	FUNCTION_BLOCK FB 303
	TITLE =G203M COUPLING DEVICE TURNER GERM 6
	//COPYRIGHT:    (C) 2009  BUHLER AG, CH-9240 UZWIL, SWITZERLAND
	//
	//PRODUCT:      WinCoS_BIW01_09
	//
	//TITLE:        COUPLING DEVICE TURNER GERM 6
	//                Machine group control
	//                Maschinengruppensteuerung
	//
	//--------------------------------------------------------------------------------
	//
	//IDENT:        AUTHOR:             DEPT:                              DATE:
	//
	//P01_FB303.1.0 K.Renz              CSB41                              13.Jan.2010
	//             1st Release
	//
	//--------------------------------------------------------------------------------
	//
	//PURPOSE:
	//
	//MANUAL :
	//
	//RESTRICTIONS:
	//
	//--------------------------------------------------------------------------------
	AUTHOR  : KR
	FAMILY  : USW
	VERSION : 9.9


	VAR
	  Gr       : FB10;	//Standard interface to group
	  InOutValue1    : DINT; //Data for user
	  InOutValue2    : DINT; //Data for user
	  OutWayConflict : BOOL;	//Data for user
	  OutSelectionOk : BOOL;	//Data for user
	  CmdNewValue : BOOL;	//Data for user
	  CmdNewJob   : BOOL;	//Data for user
	  OutCodeOK   : BOOL;	//Data for user
	  InEndOfJob  : BOOL ;	//Data for user
	  staWayOk      : BOOL ;	//Data for user
	  EdgeStartRelease : BOOL ;	//Data for user
	  USW8  : BOOL;	//Data for user
	  USW9 : BOOL;	//Data for user
	  USW10: BOOL;	//Data for user
	  USW11: BOOL;	//Data for user
	  USW12: BOOL;	//Data for user
	  USW13: BOOL;	//Data for user
	  USW14: BOOL;	//Data for user
	  USW15: BOOL;	//Data for user
	     #A_2611_MXZ21 : FB12;   // Motor
	     #A_2611_BZS22 : FB14;   // DigInpCont
	     #A_2611_BZS23 : FB14;   // DigInpCont
	     #A_2611_MXZ25 : FB12;   // Motor
	     #A_2611_BZS26 : FB14;   // DigInpCont
	     #A_2611_BZS27 : FB14;   // DigInpCont
	     #A_2611_MXZ31 : FB12;   // Motor
	     #A_2611_BZS32 : FB14;   // DigInpCont
	     #A_2611_BZS33 : FB14;   // DigInpCont
	     #A_2611_MXZ35 : FB12;   // Motor
	     #A_2611_BZS36 : FB14;   // DigInpCont
	     #A_2611_BZS37 : FB14;   // DigInpCont
	END_VAR
	VAR_TEMP
	   tmpEnable		: BOOL;
	   tmpFlag  		: BOOL;
	   tmpCmdNext		: BOOL;
	   tmpLocal  		: BOOL;
	   tmpAspOk  		: BOOL;
	   tmpHWStop 		: BOOL;
	   tmpInstanzDBNo       : INT ;
	END_VAR
	BEGIN
	NETWORK
	TITLE =
	NETWORK
	TITLE =Read command from group control
	//Parameter
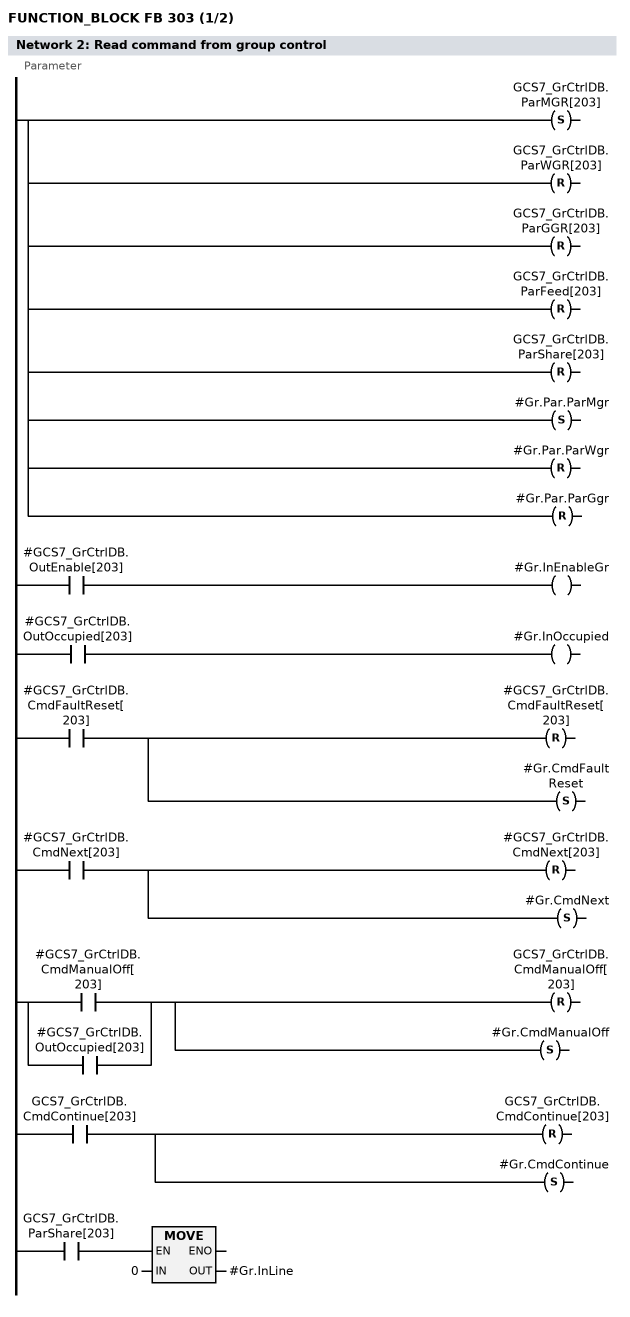
	      SET;
	      S   GCS7_GrCtrlDB.ParMGR[203];
	      R   GCS7_GrCtrlDB.ParWGR[203];
	      R   GCS7_GrCtrlDB.ParGGR[203];
	      R   GCS7_GrCtrlDB.ParFeed[203];
	      R   GCS7_GrCtrlDB.ParShare[203];
	      S   #Gr.Par.ParMgr;
	      R   #Gr.Par.ParWgr;
	      R   #Gr.Par.ParGgr;
	//Command
	      U   #GCS7_GrCtrlDB.OutEnable[203];
	      =   #Gr.InEnableGr;
	      U   #GCS7_GrCtrlDB.OutOccupied[203];
	      =   #Gr.InOccupied;
	      U   #GCS7_GrCtrlDB.CmdFaultReset[203];
	      R   #GCS7_GrCtrlDB.CmdFaultReset[203];
	      S   #Gr.CmdFaultReset;
	      U  #GCS7_GrCtrlDB.CmdNext[203];
	      R   #GCS7_GrCtrlDB.CmdNext[203];
	      S   #Gr.CmdNext;
	      U   #GCS7_GrCtrlDB.CmdManualOff[203];
	      O   #GCS7_GrCtrlDB.OutOccupied[203];
	      R   GCS7_GrCtrlDB.CmdManualOff[203];
	      S   #Gr.CmdManualOff;
	      U  GCS7_GrCtrlDB.CmdContinue[203];
	      R   GCS7_GrCtrlDB.CmdContinue[203];
	      S   #Gr.CmdContinue;
	//Init Line Number
	      U   GCS7_GrCtrlDB.ParShare[203];
	      SPBN WE00;
	      L     0;
	      T     #Gr.InLine;
	WE00: NOP   0;
	NETWORK
	TITLE =Call Methode Control
	// 1. Handle Interface PCControl
	// 2. Prepare mode --> ModePassive,ModeActive,ModeIdling
	// 3. Reset global flags of the group
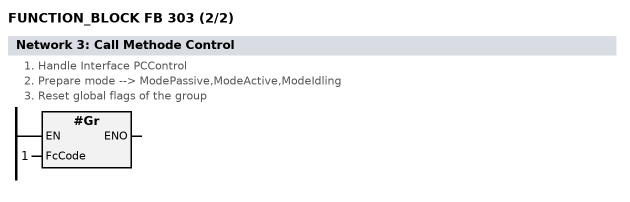
	      CALL #Gr (
	           FcCode                   := 1);
	NETWORK
	TITLE =Restart Idling Time
		L  #Gr.Par.ParIdling;
		L  2;
		>=I;
		SPB IdTm;
		T  #Gr.Par.ParIdling;
	IdTm:   NOP 0;
	      CLR;
	      S    #Gr.CmdRestartIdling;
	NETWORK
	TITLE =Prepare global flags
	NETWORK
	TITLE =Set Pattern (Target position)
	NETWORK
	TITLE =Interlocking WayOk
	//
	NETWORK
	TITLE =Interlocking Autostart
		CLR;
		R   #Gr.OutAutostart;
	NETWORK
	TITLE =Interlocking Enable
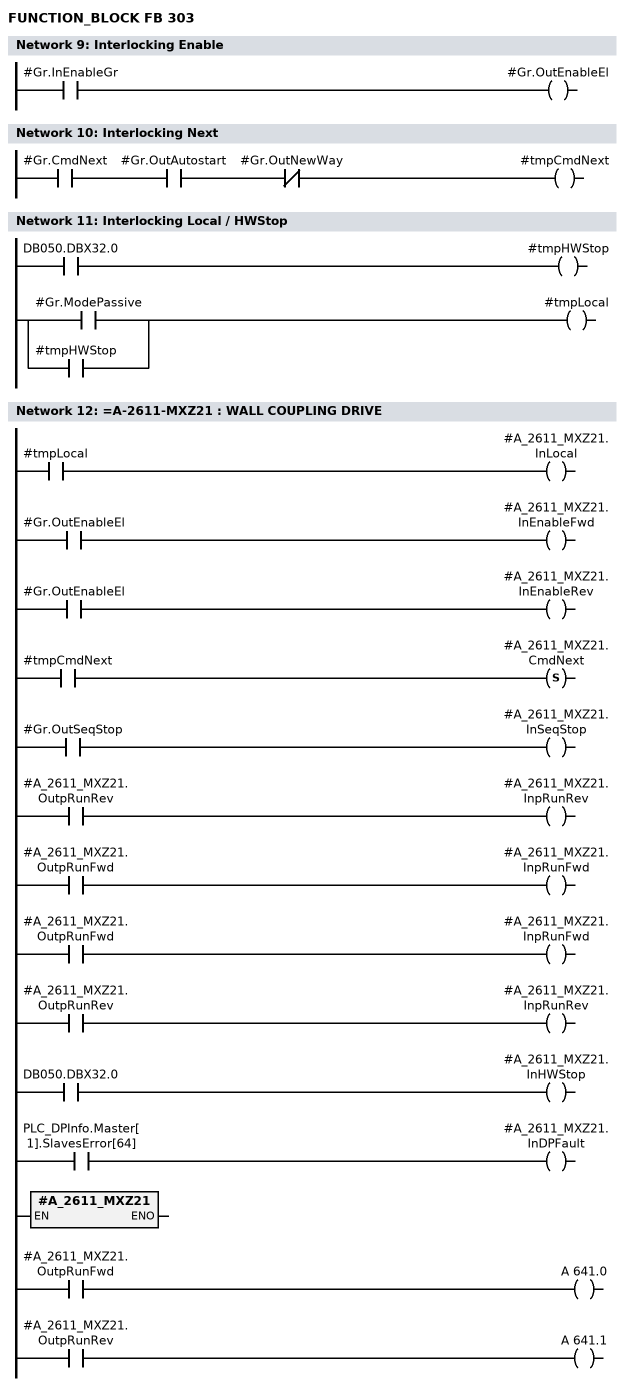
	      U     #Gr.InEnableGr;
	      =     #Gr.OutEnableEl;

	NETWORK
	TITLE =Interlocking Next
	      U     #Gr.CmdNext;
	      U     #Gr.OutAutostart;
	      UN    #Gr.OutNewWay;
	      =    #tmpCmdNext;

	NETWORK
	TITLE =Interlocking Local / HWStop
	      U    DB050.DBX32.0;
	      =    #tmpHWStop;

	      U    #Gr.ModePassive;
	      O    #tmpHWStop;
	      =    #tmpLocal;

	NETWORK
	TITLE ==A-2611-MXZ21 : WALL COUPLING DRIVE
	NOP 0;
	//-InLocal---
	      U     #tmpLocal;
	      =     #A_2611_MXZ21.InLocal;
	//
	//-Interlocking---
	      U     #Gr.OutEnableEl;
	      =     #A_2611_MXZ21.InEnableFwd;
	      U     #Gr.OutEnableEl;
	      =     #A_2611_MXZ21.InEnableRev;
	//
	      U    #tmpCmdNext;
	      S     #A_2611_MXZ21.CmdNext;
	//
	      U     #Gr.OutSeqStop;
	      =     #A_2611_MXZ21.InSeqStop;
	//
	//-Read inputs---
	      U     #A_2611_MXZ21.OutpRunRev;
	      =     #A_2611_MXZ21.InpRunRev;
	      U     #A_2611_MXZ21.OutpRunFwd;
	      =     #A_2611_MXZ21.InpRunFwd;
	      U     #A_2611_MXZ21.OutpRunFwd;
	      =     #A_2611_MXZ21.InpRunFwd;
	      U     #A_2611_MXZ21.OutpRunRev;
	      =     #A_2611_MXZ21.InpRunRev;
	      U   DB050.DBX32.0;
	      =     #A_2611_MXZ21.InHWStop;
	       U     PLC_DPInfo.Master[1].SlavesError[64];
	       =       #A_2611_MXZ21.InDPFault;
	//
	//-Set Parameters---
	//
	//-Call object control---
	      CALL  #A_2611_MXZ21;
	//
	//-Write outputs---
	      U     #A_2611_MXZ21.OutpRunFwd;
	      =     A 641.0;
	      U     #A_2611_MXZ21.OutpRunRev;
	      =     A 641.1;
	NETWORK
	TITLE ==A-2611-BZS22 : COUPLING DRIVE UNLOCKED
	NOP 0;
	//-InLocal---
	      U     #tmpLocal;
	      =     #A_2611_BZS22.InLocal;
	//
	//-Monitoring---
	      CLR;
	      =      #A_2611_BZS22.InMonTrue;
	      CLR;
	      =      #A_2611_BZS22.InMonFalse;
	//
	//-PreAlarm---
	      CLR;
	      =      #A_2611_BZS22.InPreAlarmTrue;
	      CLR;
	      =      #A_2611_BZS22.InPreAlarmFalse;
	//
	//-Additional commands---
	//      CLR
	//      S     #A_2611_BZS22.CmdRunTimeOutTime
	//
	//-Read inputs---
	      U     E 643.0;
	      =     #A_2611_BZS22.InpTrue;
	      U   DB050.DBX32.0;
	      =     #A_2611_BZS22.InHWStop;
	       U     PLC_DPInfo.Master[1].SlavesError[64];
	       =       #A_2611_BZS22.InDPFault;
	//
	//-Set Parameters---
	//
	//-Call object control---
	      CALL  #A_2611_BZS22;
	//
	//-Write outputs---
	NETWORK
	TITLE ==A-2611-BZS23 : COUPLING DRIVE LOCKED
	NOP 0;
	//-InLocal---
	      U     #tmpLocal;
	      =     #A_2611_BZS23.InLocal;
	//
	//-Monitoring---
	      CLR;
	      =      #A_2611_BZS23.InMonTrue;
	      CLR;
	      =      #A_2611_BZS23.InMonFalse;
	//
	//-PreAlarm---
	      CLR;
	      =      #A_2611_BZS23.InPreAlarmTrue;
	      CLR;
	      =      #A_2611_BZS23.InPreAlarmFalse;
	//
	//-Additional commands---
	//      CLR
	//      S     #A_2611_BZS23.CmdRunTimeOutTime
	//
	//-Read inputs---
	      U     E 643.1;
	      =     #A_2611_BZS23.InpTrue;
	      U   DB050.DBX32.0;
	      =     #A_2611_BZS23.InHWStop;
	       U     PLC_DPInfo.Master[1].SlavesError[64];
	       =       #A_2611_BZS23.InDPFault;
	//
	//-Set Parameters---
	//
	//-Call object control---
	      CALL  #A_2611_BZS23;
	//
	//-Write outputs---
	NETWORK
	TITLE ==A-2611-MXZ25 : WALL COUPLING DRIVE
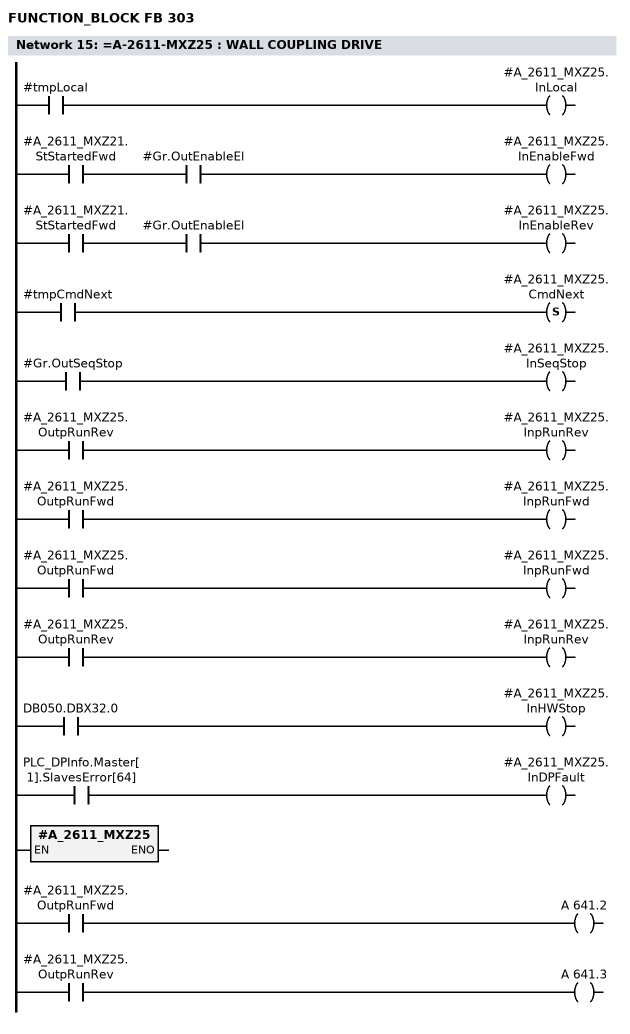
	NOP 0;
	//-InLocal---
	      U     #tmpLocal;
	      =     #A_2611_MXZ25.InLocal;
	//
	//-Interlocking---
	      U     #A_2611_MXZ21.StStartedFwd;
	      U     #Gr.OutEnableEl;
	      =     #A_2611_MXZ25.InEnableFwd;
	      U     #A_2611_MXZ21.StStartedFwd;
	      U     #Gr.OutEnableEl;
	      =     #A_2611_MXZ25.InEnableRev;
	//
	      U    #tmpCmdNext;
	      S     #A_2611_MXZ25.CmdNext;
	//
	      U     #Gr.OutSeqStop;
	      =     #A_2611_MXZ25.InSeqStop;
	//
	//-Read inputs---
	      U     #A_2611_MXZ25.OutpRunRev;
	      =     #A_2611_MXZ25.InpRunRev;
	      U     #A_2611_MXZ25.OutpRunFwd;
	      =     #A_2611_MXZ25.InpRunFwd;
	      U     #A_2611_MXZ25.OutpRunFwd;
	      =     #A_2611_MXZ25.InpRunFwd;
	      U     #A_2611_MXZ25.OutpRunRev;
	      =     #A_2611_MXZ25.InpRunRev;
	      U   DB050.DBX32.0;
	      =     #A_2611_MXZ25.InHWStop;
	       U     PLC_DPInfo.Master[1].SlavesError[64];
	       =       #A_2611_MXZ25.InDPFault;
	//
	//-Set Parameters---
	//
	//-Call object control---
	      CALL  #A_2611_MXZ25;
	//
	//-Write outputs---
	      U     #A_2611_MXZ25.OutpRunFwd;
	      =     A 641.2;
	      U     #A_2611_MXZ25.OutpRunRev;
	      =     A 641.3;
	NETWORK
	TITLE ==A-2611-BZS26 : COUPLING DRIVE UNLOCKED
	NOP 0;
	//-InLocal---
	      U     #tmpLocal;
	      =     #A_2611_BZS26.InLocal;
	//
	//-Monitoring---
	      CLR;
	      =      #A_2611_BZS26.InMonTrue;
	      CLR;
	      =      #A_2611_BZS26.InMonFalse;
	//
	//-PreAlarm---
	      CLR;
	      =      #A_2611_BZS26.InPreAlarmTrue;
	      CLR;
	      =      #A_2611_BZS26.InPreAlarmFalse;
	//
	//-Additional commands---
	//      CLR
	//      S     #A_2611_BZS26.CmdRunTimeOutTime
	//
	//-Read inputs---
	      U     E 643.2;
	      =     #A_2611_BZS26.InpTrue;
	      U   DB050.DBX32.0;
	      =     #A_2611_BZS26.InHWStop;
	       U     PLC_DPInfo.Master[1].SlavesError[64];
	       =       #A_2611_BZS26.InDPFault;
	//
	//-Set Parameters---
	//
	//-Call object control---
	      CALL  #A_2611_BZS26;
	//
	//-Write outputs---
	NETWORK
	TITLE ==A-2611-BZS27 : COUPLING DRIVE LOCKED
	NOP 0;
	//-InLocal---
	      U     #tmpLocal;
	      =     #A_2611_BZS27.InLocal;
	//
	//-Monitoring---
	      CLR;
	      =      #A_2611_BZS27.InMonTrue;
	      CLR;
	      =      #A_2611_BZS27.InMonFalse;
	//
	//-PreAlarm---
	      CLR;
	      =      #A_2611_BZS27.InPreAlarmTrue;
	      CLR;
	      =      #A_2611_BZS27.InPreAlarmFalse;
	//
	//-Additional commands---
	//      CLR
	//      S     #A_2611_BZS27.CmdRunTimeOutTime
	//
	//-Read inputs---
	      U     E 643.3;
	      =     #A_2611_BZS27.InpTrue;
	      U   DB050.DBX32.0;
	      =     #A_2611_BZS27.InHWStop;
	       U     PLC_DPInfo.Master[1].SlavesError[64];
	       =       #A_2611_BZS27.InDPFault;
	//
	//-Set Parameters---
	//
	//-Call object control---
	      CALL  #A_2611_BZS27;
	//
	//-Write outputs---
	NETWORK
	TITLE ==A-2611-MXZ31 : WALL COUPLING DRIVE
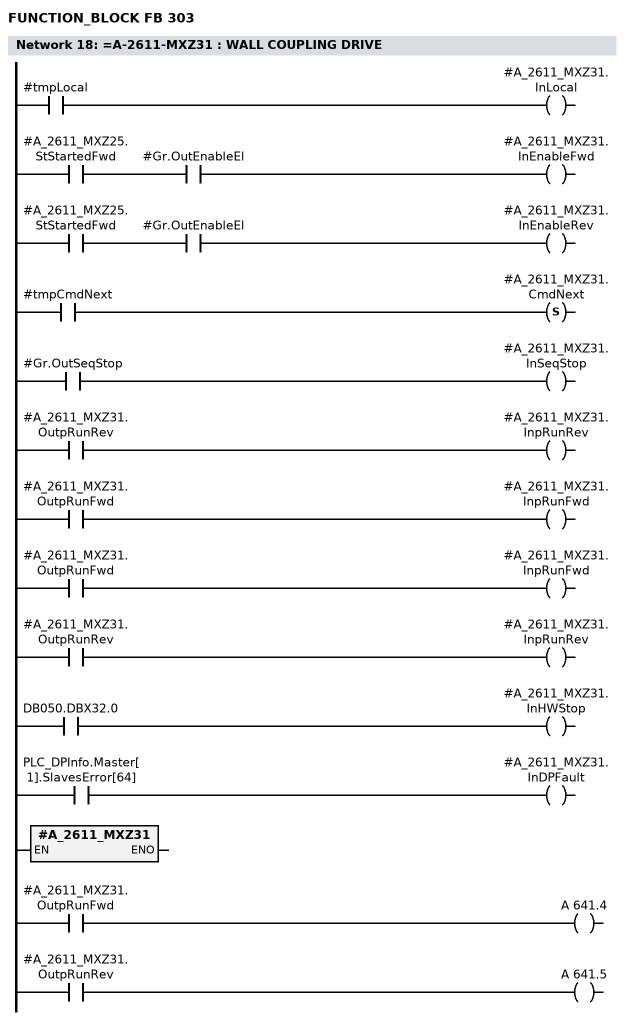
	NOP 0;
	//-InLocal---
	      U     #tmpLocal;
	      =     #A_2611_MXZ31.InLocal;
	//
	//-Interlocking---
	      U     #A_2611_MXZ25.StStartedFwd;
	      U     #Gr.OutEnableEl;
	      =     #A_2611_MXZ31.InEnableFwd;
	      U     #A_2611_MXZ25.StStartedFwd;
	      U     #Gr.OutEnableEl;
	      =     #A_2611_MXZ31.InEnableRev;
	//
	      U    #tmpCmdNext;
	      S     #A_2611_MXZ31.CmdNext;
	//
	      U     #Gr.OutSeqStop;
	      =     #A_2611_MXZ31.InSeqStop;
	//
	//-Read inputs---
	      U     #A_2611_MXZ31.OutpRunRev;
	      =     #A_2611_MXZ31.InpRunRev;
	      U     #A_2611_MXZ31.OutpRunFwd;
	      =     #A_2611_MXZ31.InpRunFwd;
	      U     #A_2611_MXZ31.OutpRunFwd;
	      =     #A_2611_MXZ31.InpRunFwd;
	      U     #A_2611_MXZ31.OutpRunRev;
	      =     #A_2611_MXZ31.InpRunRev;
	      U   DB050.DBX32.0;
	      =     #A_2611_MXZ31.InHWStop;
	       U     PLC_DPInfo.Master[1].SlavesError[64];
	       =       #A_2611_MXZ31.InDPFault;
	//
	//-Set Parameters---
	//
	//-Call object control---
	      CALL  #A_2611_MXZ31;
	//
	//-Write outputs---
	      U     #A_2611_MXZ31.OutpRunFwd;
	      =     A 641.4;
	      U     #A_2611_MXZ31.OutpRunRev;
	      =     A 641.5;
	NETWORK
	TITLE ==A-2611-BZS32 : COUPLING DRIVE UNLOCKED
	NOP 0;
	//-InLocal---
	      U     #tmpLocal;
	      =     #A_2611_BZS32.InLocal;
	//
	//-Monitoring---
	      CLR;
	      =      #A_2611_BZS32.InMonTrue;
	      CLR;
	      =      #A_2611_BZS32.InMonFalse;
	//
	//-PreAlarm---
	      CLR;
	      =      #A_2611_BZS32.InPreAlarmTrue;
	      CLR;
	      =      #A_2611_BZS32.InPreAlarmFalse;
	//
	//-Additional commands---
	//      CLR
	//      S     #A_2611_BZS32.CmdRunTimeOutTime
	//
	//-Read inputs---
	      U     E 643.4;
	      =     #A_2611_BZS32.InpTrue;
	      U   DB050.DBX32.0;
	      =     #A_2611_BZS32.InHWStop;
	       U     PLC_DPInfo.Master[1].SlavesError[64];
	       =       #A_2611_BZS32.InDPFault;
	//
	//-Set Parameters---
	//
	//-Call object control---
	      CALL  #A_2611_BZS32;
	//
	//-Write outputs---
	NETWORK
	TITLE ==A-2611-BZS33 : COUPLING DRIVE LOCKED
	NOP 0;
	//-InLocal---
	      U     #tmpLocal;
	      =     #A_2611_BZS33.InLocal;
	//
	//-Monitoring---
	      CLR;
	      =      #A_2611_BZS33.InMonTrue;
	      CLR;
	      =      #A_2611_BZS33.InMonFalse;
	//
	//-PreAlarm---
	      CLR;
	      =      #A_2611_BZS33.InPreAlarmTrue;
	      CLR;
	      =      #A_2611_BZS33.InPreAlarmFalse;
	//
	//-Additional commands---
	//      CLR
	//      S     #A_2611_BZS33.CmdRunTimeOutTime
	//
	//-Read inputs---
	      U     E 643.5;
	      =     #A_2611_BZS33.InpTrue;
	      U   DB050.DBX32.0;
	      =     #A_2611_BZS33.InHWStop;
	       U     PLC_DPInfo.Master[1].SlavesError[64];
	       =       #A_2611_BZS33.InDPFault;
	//
	//-Set Parameters---
	//
	//-Call object control---
	      CALL  #A_2611_BZS33;
	//
	//-Write outputs---
	NETWORK
	TITLE ==A-2611-MXZ35 : WALL COUPLING DRIVE
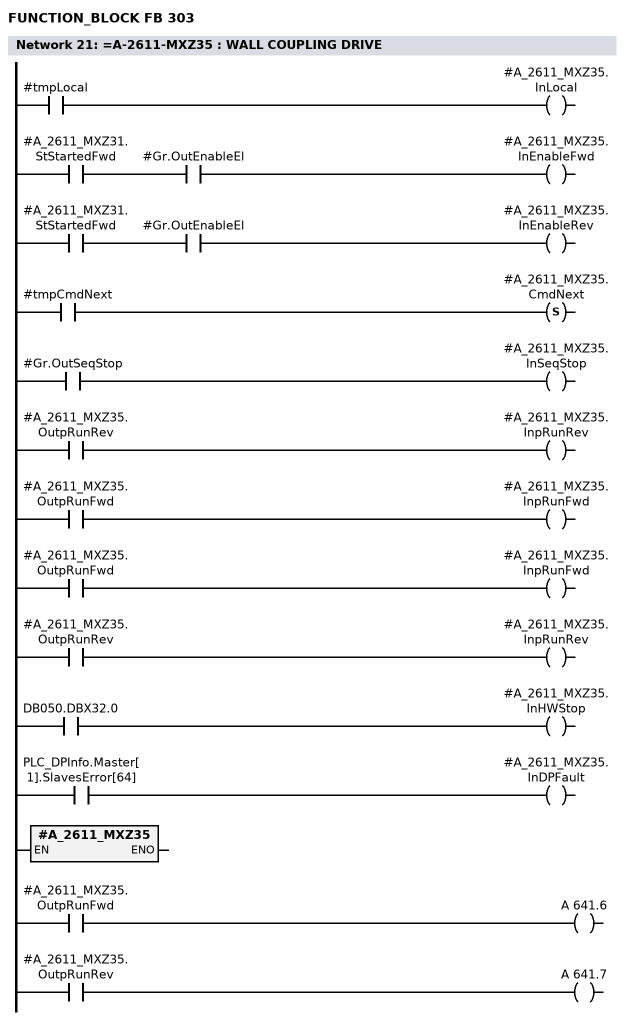
	NOP 0;
	//-InLocal---
	      U     #tmpLocal;
	      =     #A_2611_MXZ35.InLocal;
	//
	//-Interlocking---
	      U     #A_2611_MXZ31.StStartedFwd;
	      U     #Gr.OutEnableEl;
	      =     #A_2611_MXZ35.InEnableFwd;
	      U     #A_2611_MXZ31.StStartedFwd;
	      U     #Gr.OutEnableEl;
	      =     #A_2611_MXZ35.InEnableRev;
	//
	      U    #tmpCmdNext;
	      S     #A_2611_MXZ35.CmdNext;
	//
	      U     #Gr.OutSeqStop;
	      =     #A_2611_MXZ35.InSeqStop;
	//
	//-Read inputs---
	      U     #A_2611_MXZ35.OutpRunRev;
	      =     #A_2611_MXZ35.InpRunRev;
	      U     #A_2611_MXZ35.OutpRunFwd;
	      =     #A_2611_MXZ35.InpRunFwd;
	      U     #A_2611_MXZ35.OutpRunFwd;
	      =     #A_2611_MXZ35.InpRunFwd;
	      U     #A_2611_MXZ35.OutpRunRev;
	      =     #A_2611_MXZ35.InpRunRev;
	      U   DB050.DBX32.0;
	      =     #A_2611_MXZ35.InHWStop;
	       U     PLC_DPInfo.Master[1].SlavesError[64];
	       =       #A_2611_MXZ35.InDPFault;
	//
	//-Set Parameters---
	//
	//-Call object control---
	      CALL  #A_2611_MXZ35;
	//
	//-Write outputs---
	      U     #A_2611_MXZ35.OutpRunFwd;
	      =     A 641.6;
	      U     #A_2611_MXZ35.OutpRunRev;
	      =     A 641.7;
	NETWORK
	TITLE ==A-2611-BZS36 : COUPLING DRIVE UNLOCKED
	NOP 0;
	//-InLocal---
	      U     #tmpLocal;
	      =     #A_2611_BZS36.InLocal;
	//
	//-Monitoring---
	      CLR;
	      =      #A_2611_BZS36.InMonTrue;
	      CLR;
	      =      #A_2611_BZS36.InMonFalse;
	//
	//-PreAlarm---
	      CLR;
	      =      #A_2611_BZS36.InPreAlarmTrue;
	      CLR;
	      =      #A_2611_BZS36.InPreAlarmFalse;
	//
	//-Additional commands---
	//      CLR
	//      S     #A_2611_BZS36.CmdRunTimeOutTime
	//
	//-Read inputs---
	      U     E 643.6;
	      =     #A_2611_BZS36.InpTrue;
	      U   DB050.DBX32.0;
	      =     #A_2611_BZS36.InHWStop;
	       U     PLC_DPInfo.Master[1].SlavesError[64];
	       =       #A_2611_BZS36.InDPFault;
	//
	//-Set Parameters---
	//
	//-Call object control---
	      CALL  #A_2611_BZS36;
	//
	//-Write outputs---
	NETWORK
	TITLE ==A-2611-BZS37 : COUPLING DRIVE LOCKED
	NOP 0;
	//-InLocal---
	      U     #tmpLocal;
	      =     #A_2611_BZS37.InLocal;
	//
	//-Monitoring---
	      CLR;
	      =      #A_2611_BZS37.InMonTrue;
	      CLR;
	      =      #A_2611_BZS37.InMonFalse;
	//
	//-PreAlarm---
	      CLR;
	      =      #A_2611_BZS37.InPreAlarmTrue;
	      CLR;
	      =      #A_2611_BZS37.InPreAlarmFalse;
	//
	//-Additional commands---
	//      CLR
	//      S     #A_2611_BZS37.CmdRunTimeOutTime
	//
	//-Read inputs---
	      U     E 643.7;
	      =     #A_2611_BZS37.InpTrue;
	      U   DB050.DBX32.0;
	      =     #A_2611_BZS37.InHWStop;
	       U     PLC_DPInfo.Master[1].SlavesError[64];
	       =       #A_2611_BZS37.InDPFault;
	//
	//-Set Parameters---
	//
	//-Call object control---
	      CALL  #A_2611_BZS37;
	//
	//-Write outputs---
	NETWORK
	TITLE =Test Fault
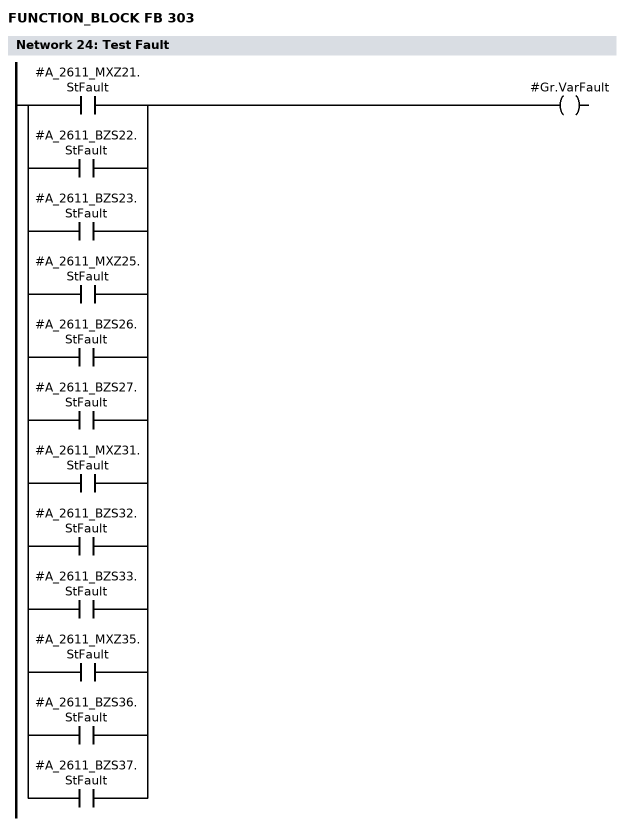
	      U     #A_2611_MXZ21.StFault;
	      O     #A_2611_BZS22.StFault;
	      O     #A_2611_BZS23.StFault;
	      O     #A_2611_MXZ25.StFault;
	      O     #A_2611_BZS26.StFault;
	      O     #A_2611_BZS27.StFault;
	      O     #A_2611_MXZ31.StFault;
	      O     #A_2611_BZS32.StFault;
	      O     #A_2611_BZS33.StFault;
	      O     #A_2611_MXZ35.StFault;
	      O     #A_2611_BZS36.StFault;
	      O     #A_2611_BZS37.StFault;
	      =     #Gr.VarFault;
	NETWORK
	TITLE =Test Warning
	      CLR;
	      =     #Gr.OutWarning;
	NETWORK
	TITLE =Test Stopped
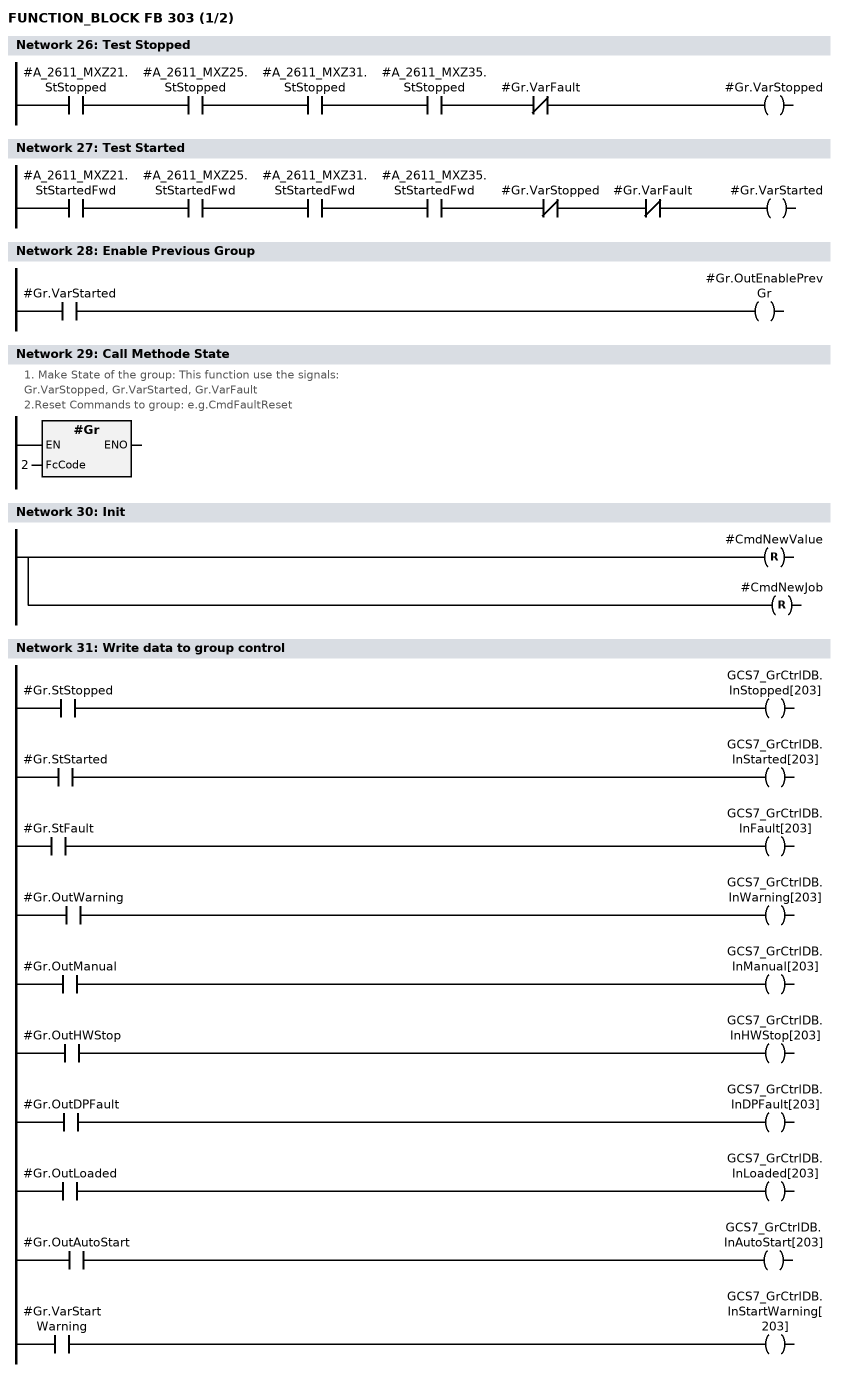
	      U     #A_2611_MXZ21.StStopped;
	      U     #A_2611_MXZ25.StStopped;
	      U     #A_2611_MXZ31.StStopped;
	      U     #A_2611_MXZ35.StStopped;
	      UN   #Gr.VarFault;
	      =     #Gr.VarStopped;
	NETWORK
	TITLE =Test Started
	      U     #A_2611_MXZ21.StStartedFwd;
	      U     #A_2611_MXZ25.StStartedFwd;
	      U     #A_2611_MXZ31.StStartedFwd;
	      U     #A_2611_MXZ35.StStartedFwd;
	      UN  #Gr.VarStopped;
	      UN  #Gr.VarFault;
	      =     #Gr.VarStarted;
	NETWORK
	TITLE =Enable Previous Group
	      U    #Gr.VarStarted;
	      =     #Gr.OutEnablePrevGr;
	NETWORK
	TITLE =Call Methode State
	//1. Make State of the group: This function use the signals:
	//        Gr.VarStopped, Gr.VarStarted, Gr.VarFault
	//2.Reset Commands to group: e.g.CmdFaultReset
	      CALL #Gr (
	           FcCode                   := 2);
	NETWORK
	TITLE =Init
	      SET;
	      R    #CmdNewValue;
	      R    #CmdNewJob;
	NETWORK
	TITLE =Write data to group control
	      U   #Gr.StStopped;
	      =   GCS7_GrCtrlDB.InStopped[203];
	      U   #Gr.StStarted;
	      =   GCS7_GrCtrlDB.InStarted[203];
	      U   #Gr.StFault;
	      =   GCS7_GrCtrlDB.InFault[203];
	      U   #Gr.OutWarning;
	      =   GCS7_GrCtrlDB.InWarning[203];
	      U   #Gr.OutManual;
	      =   GCS7_GrCtrlDB.InManual[203];
	      U   #Gr.OutHWStop;
	      =   GCS7_GrCtrlDB.InHWStop[203];
	      U   #Gr.OutDPFault;
	      =   GCS7_GrCtrlDB.InDPFault[203];
	      U   #Gr.OutLoaded;
	      =   GCS7_GrCtrlDB.InLoaded[203];
	      U   #Gr.OutAutoStart;
	      =   GCS7_GrCtrlDB.InAutoStart[203];
	      U   #Gr.VarStartWarning;
	      =   GCS7_GrCtrlDB.InStartWarning[203];
	NETWORK
	TITLE =End of block
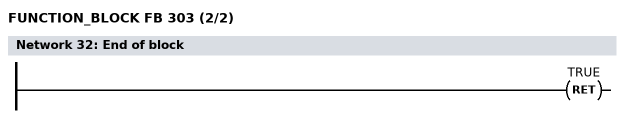

	BE

	END_FUNCTION_BLOCK
